FUNCTION_BLOCK FB3_XmlSvrRW_Recipe
VAR_INPUT
	bWriteSt				: BOOL;
	bReadSt					: BOOL;
	bShutdownRequestFlag 	: BOOL;

	eVariableType			: E_XMLVariableType;
	eXmlRwMode				: E_XmlRWMode;
		
	sDefaultFilePath		: STRING := 'C:\JKS\PLC\XML\';
	sFileExtension			: STRING := 'XML';
	
END_VAR
VAR_OUTPUT
	bWrite_Done				: BOOL;
	bWrite_Busy				: BOOL;
	bWrite_Error			: BOOL;
	udWrite_ErrId			: UDINT;
	bRead_Done				: BOOL;
	bRead_Busy				: BOOL;
	bRead_Error				: BOOL;
	udRead_ErrId 			: UDINT;
	bReadyToShutdownFlag 	: BOOL;
	sErrorMessage			: STRING;
	iTotalTime_100ms		: INT;
	iExportedImportedQty	: INT;
	iProgressPercentage		: INT;
END_VAR

VAR
		fbXmlSrvWriteByAdd	: FB_XmlSrvWrite;
		fbXmlSrvReadByAdd	: FB_XmlSrvRead;
		fbFileDelete		: FB_FileDelete;
	bWriteStRE						: R_TRIG;
	bReadStRE						: R_TRIG;
	iArrayId_ProRepRecipeQty		: INT;
	iArrayId_iSSERRecipeQty			: INT;
	iArrayId_iSSURRecipeQty			: INT;
	iArrayId_iSSMRRecipeQty			: INT;
	iArrayId_SSERProcessStnQty		: INT;
	iArrayId_SSURProcessStnQty		: INT;
	iArrayId_SSMRProcessStnQty		: INT;
	iFL								: INT;
	iCase							: INT;
	bFound							: BOOL;

	bWriteSt_Int					: BOOL;
	bReadSt_Int						: BOOL;
	bWrite_Busy_Int					: BOOL;
	bRead_Busy_Int					: BOOL;
	bFileDeleteSt					: BOOL;
	sFilePath_Int					: T_MaxString;
	sXPath_Int						: T_MaxString;

	
	iRepType			: INT;
	
	
	pSymAddr_Int		: PVOID;
	pSymAddr_Empty		: PVOID;

	cbSymSize_Int		: UDINT;
	sFileName_Main			: STRING;
	sFileName_Sub1			: STRING;
	sFileName_Sub2			: STRING;

	sXPath_Main			: STRING; 	// No Spacing is allowed
	sXPath_Sub1			: STRING;	// No Spacing is allowed
	sXPath_Sub2			: STRING;	// No Spacing is allowed

	
	bRead_Error_Int: BOOL;
	iTotalWriteTask: INT;
	iProRepTask: INT;
	iSSERTask: INT;
	iSSURTask: INT;
	iSSMRTask: INT;
END_VAR


IF NOT bWriteSt AND NOT bReadSt THEN
	iCase 	:= 0;
END_IF

bWriteStRE(CLK	:=bWriteSt AND NOT bShutdownRequestFlag 	, Q=> );
bReadStRE(CLK	:=bReadSt AND NOT bShutdownRequestFlag  	, Q=> );


// Shutdown request control
	bReadyToShutdownFlag := NOT bWrite_Busy AND NOT bRead_Busy AND bShutdownRequestFlag;


// Capture Total Time for Read or Write
IF iCase = 1 OR (iCase >= 10 AND iCase < 19) OR (iCase >= 20 AND iCase < 29) THEN
	IF bClockPulse_0_1Sec THEN
		iTotalTime_100ms := iTotalTime_100ms + 1;
	END_IF
END_IF


fbXmlSrvWriteByAdd(
	sNetId			:= '', 
	ePath			:= PATH_GENERIC, 
	nMode			:= XMLSRV_ADDMISSING, 
	pSymAddr		:= pSymAddr_Int, 
	cbSymSize		:= cbSymSize_Int, 
	sFilePath		:= sFilePath_Int, 
	sXPath			:= sXPath_Int, 
	bExecute		:= bWriteSt_Int, 
	tTimeout		:= T#5S, 
	bBusy			=> bWrite_Busy_Int, 
	bError			=> bWrite_Error);

fbXmlSrvReadByAdd(
	sNetId			:= '', 
	ePath			:= PATH_GENERIC, 
	nMode			:= XMLSRV_SKIPMISSING, 
	pSymAddr		:= pSymAddr_Int, 
	cbSymSize		:= cbSymSize_Int, 
	sFilePath		:= sFilePath_Int, 
	sXPath			:= sXPath_Int, 
	bExecute		:= bReadSt_Int, 
	tTimeout		:= T#5S, 
	bBusy			=> bRead_Busy_Int, 
	bError			=> bRead_Error_Int, 
	nErrId			=> );

IF 		bWriteStRE.Q 	AND NOT bReadSt 	AND NOT bRead_Busy 	THEN 	iCase := 1; 	bWrite_Busy := TRUE;
ELSIF	bReadStRE.Q		AND NOT bWriteSt 	AND NOT bWrite_Busy	THEN 	iCase := 1;		bRead_Busy := TRUE;			END_IF	

IF bRead_Error_Int AND fbXmlSrvReadByAdd.nErrId <> 1804 THEN
	bRead_Error := TRUE;
ELSE	
	bRead_Error := FALSE;
END_IF

CASE iCase OF
	
	0: 	// Reset ALL

			iArrayId_ProRepRecipeQty		:= 0;
			iArrayId_iSSERRecipeQty			:= 0;
			iArrayId_iSSURRecipeQty			:= 0;
			iArrayId_iSSMRRecipeQty			:= 0;
			iArrayId_SSERProcessStnQty		:= 0;
			iArrayId_SSURProcessStnQty		:= 0;
			iArrayId_SSMRProcessStnQty		:= 0;

			udWrite_ErrId			:= 0;
			bWrite_Busy				:= FALSE;
			bWrite_Error			:= FALSE;
			bWrite_Done				:= FALSE;

			udRead_ErrId			:= 0;
			bRead_Busy				:= FALSE;
			bRead_Error				:= FALSE;
			bRead_Done				:= FALSE;
	
			
			iTotalTime_100ms		:= 0;	

			bWriteSt_Int 			:= FALSE;
			bReadSt_Int 			:= FALSE;
			bFileDeleteSt			:= FALSE;
		
			iExportedImportedQty	:= 0;			
			pSymAddr_Int			:= pSymAddr_Empty;
			cbSymSize_Int			:= 0;	
			sFilePath_Int			:= '';
			sXPath_Int				:= '';	
			
			iRepType				:= 0;   // 1: Product Recipe, 2: SSER, 3: SSUR, 4: SSMR

			
			
			
	1: // Check Avaiable Array to trigger Read/Write

			IF iRepType 					< 1 	THEN iRepType 						:= 1; 	END_IF
			IF iArrayId_ProRepRecipeQty		< 1 	THEN iArrayId_ProRepRecipeQty	 	:= 1;	END_IF
			IF iArrayId_SSERProcessStnQty 	< 1 	THEN iArrayId_SSERProcessStnQty 	:= 1;	END_IF
			IF iArrayId_iSSERRecipeQty 		< 1	 	THEN iArrayId_iSSERRecipeQty 		:= 1; 	END_IF			
			IF iArrayId_SSURProcessStnQty 	< 1 	THEN iArrayId_SSURProcessStnQty 	:= 1;	END_IF
			IF iArrayId_iSSURRecipeQty 		< 1	 	THEN iArrayId_iSSURRecipeQty 		:= 1; 	END_IF
			IF iArrayId_SSMRProcessStnQty 	< 1 	THEN iArrayId_SSMRProcessStnQty 	:= 1;	END_IF
			IF iArrayId_iSSMRRecipeQty 		< 1	 	THEN iArrayId_iSSMRRecipeQty 		:= 1; 	END_IF
				
			CASE eXmlRwMode OF 
			
(*				eXmlMode_MergeAllByType:
						acMergeAllByType();							// ACTION			
*)						
				eXmlMode_SeperateByProductAndStation:			
						acSeperateByProductAndStation();			// ACTION
			
(*				eXmlMode_SeperateAll:			
						acSeperateAll();							// ACTION
*)
			END_CASE

						acGenerate_Filename_XPath();				// ACTION		
		
			IF 		bWrite_Busy AND iCase <> 19 THEN		
					iCase 	:= 12;					
			
			ELSIF 	bRead_Busy AND iCase <> 29 THEN		
					iCase 	:= 22;					
			END_IF			

				
	12: // Write Start

			bWriteSt_Int := TRUE;
	
			IF fbXmlSrvWriteByAdd.bExecute AND NOT fbXmlSrvWriteByAdd.bBusy AND NOT fbXmlSrvWriteByAdd.bError 
			AND 	fbXmlSrvWriteByAdd.pSymAddr		= pSymAddr_Int
			AND 	fbXmlSrvWriteByAdd.cbSymSize	= cbSymSize_Int	
			AND 	fbXmlSrvWriteByAdd.sFilePath 	= sFilePath_Int
			AND 	fbXmlSrvWriteByAdd.sXPath		= sXPath_Int		
			THEN	iCase := 13; // Write Done -> Proceed to clear FB to prepare for Next Cycle (Array) 
					iExportedImportedQty := iExportedImportedQty + 1;			
				
			ELSIF fbXmlSrvWriteByAdd.bExecute AND fbXmlSrvWriteByAdd.bError THEN
				udWrite_ErrId := fbXmlSrvWriteByAdd.nErrId;
				mtLogErrorId();
				iCase := 99;	// WRITE ERROR

				
			END_IF

	13: 	//  Write - prepare for Next Cycle (Array) 
			
			bWriteSt_Int := FALSE;
	
			IF NOT fbXmlSrvWriteByAdd.bExecute AND NOT fbXmlSrvWriteByAdd.bBusy  THEN
				iCase := 1; // Proceed to Next Cycle (Array) 
			END_IF
		
		
	19: // Write - All Done 
		
			bWrite_Busy 	:= FALSE;
			bWrite_Done 	:= TRUE;
			
	22: // Read Start

			bReadSt_Int := TRUE;
	
			IF 		fbXmlSrvReadByAdd.bExecute AND NOT fbXmlSrvReadByAdd.bBusy AND NOT fbXmlSrvReadByAdd.bError 
			AND 	fbXmlSrvReadByAdd.pSymAddr		= pSymAddr_Int
			AND 	fbXmlSrvReadByAdd.cbSymSize		= cbSymSize_Int
			AND 	fbXmlSrvReadByAdd.sFilePath 	= sFilePath_Int
			AND 	fbXmlSrvReadByAdd.sXPath		= sXPath_Int		
			THEN	iCase := 23; bFileDeleteSt := TRUE;	// Read Done -> Proceed to delete file and clear FB to prepare for Next Cycle (Array)			
					iExportedImportedQty := iExportedImportedQty + 1;			

			ELSIF fbXmlSrvReadByAdd.bExecute AND fbXmlSrvReadByAdd.bError AND fbXmlSrvReadByAdd.nErrId = 1804 
			THEN	iCase := 23; // Object Not Found -> Skipped and Proceed to clear FB to prepare for Next Cycle (Array)		
					
			ELSIF fbXmlSrvReadByAdd.bExecute AND fbXmlSrvReadByAdd.bError THEN
				udRead_ErrId := fbXmlSrvReadByAdd.nErrId;
				mtLogErrorId();
				iCase := 99;	// READ ERROR
			END_IF

	23:		// Delete file after read
			fbFileDelete(
			sNetId			:= '', 
			sPathName		:= sFilePath_Int, 
			ePath			:= PATH_GENERIC, 
			bExecute		:= bFileDeleteSt, 
			tTimeout		:= T#2S, 
			bBusy			=> , 
			bError			=> , 
			nErrId			=> );		

			IF fbFileDelete.bExecute AND NOT fbFileDelete.bBusy THEN
				bFileDeleteSt := FALSE;
			END_IF

			IF NOT fbFileDelete.bExecute AND NOT bFileDeleteSt THEN
				iCase := 24;	// Delete file done, proceed to clear FB to prepare for Next Cycle (Array)
			END_IF
			
	24: 	//  Read - prepare for Next Cycle (Array) 
			
			bReadSt_Int := FALSE;
	
			IF NOT fbXmlSrvReadByAdd.bExecute AND NOT fbXmlSrvReadByAdd.bBusy  THEN
				iCase := 1; // Proceed to Next Cycle (Array)
			END_IF
		
		
	29: // Read - All Done 
		
			bRead_Busy 	:= FALSE;
			bRead_Done 	:= TRUE;
		
	
	99: // Error
	
			bWriteSt_Int 	:= FALSE;
			bReadSt_Int 	:= FALSE;

END_CASE

// Progress Percentage
		IF NOT bWriteSt AND NOT bReadSt  THEN
			iProgressPercentage := 0;			

		ELSIF (bWriteSt AND NOT bWrite_Done) OR (bReadSt AND NOT bRead_Done) THEN
			acProgressPercentage();
		
		ELSIF (bWriteSt AND bWrite_Done) OR (bReadSt AND bRead_Done) THEN
			iProgressPercentage := 100;			
		END_IF

ACTION acGenerate_Filename_XPath:

		IF 		bWrite_Busy THEN		
		sFilePath_Int	:=	concat(sDefaultFilePath,	'Manual_Export'	);
		sFilePath_Int	:=	concat(sFilePath_Int,		'\'				);
		sFilePath_Int	:=	concat(sFilePath_Int,		sFileName_Main	);
		
		ELSIF 	bRead_Busy THEN		
		sFilePath_Int	:=	concat(sDefaultFilePath,	'Manual_Import'	);
		sFilePath_Int	:=	concat(sFilePath_Int,		'\'				);
		sFilePath_Int	:=	concat(sFilePath_Int,		sFileName_Main	);
		END_IF			
	
		IF sFileName_Sub1 <> '' THEN
		sFilePath_Int	:=	concat(sFilePath_Int,		'_'				);
		sFilePath_Int	:=	concat(sFilePath_Int,		sFileName_Sub1	);
		END_IF
		
		IF sFileName_Sub2 <> '' THEN
		sFilePath_Int	:=	concat(sFilePath_Int,		'_'				);
		sFilePath_Int	:=	concat(sFilePath_Int,		sFileName_Sub2	);
		END_IF
		
		sFilePath_Int	:=	concat(sFilePath_Int,		'.'				);
		sFilePath_Int	:=	concat(sFilePath_Int,		sFileExtension	);


							
		sXPath_Int		:=	concat('/Recipe/',		sXPath_Main		);

		IF sXPath_Sub1 <> '' THEN
		sXPath_Int		:=	concat(sXPath_Int,		'/ID'			);
		sXPath_Int		:=	concat(sXPath_Int,		sXPath_Sub1		);
		END_IF
		
		IF sXPath_Sub2 <> '' THEN
		sXPath_Int		:=	concat(sXPath_Int,		'/ID'			);
		sXPath_Int		:=	concat(sXPath_Int,		sXPath_Sub2		);
		END_IF
END_ACTION

ACTION acMergeAllByType:

	IF 		iRepType 		= eXmlParTypeSSER                       
	THEN	pSymAddr_Int 	:= ADR	(fbMainStationProcess_Stn);  
			cbSymSize_Int	:= SIZEOF(fbMainStationProcess_Stn);
			sFileName_Main	:= 'MergeAll\SSER';                 
			sFileName_Sub1	:= 'All';                           
			sFileName_Sub2	:= '';                              
			sXPath_Main		:= 'AR2dsSSER';                       
			sXPath_Sub1		:= '';                                
			sXPath_Sub2		:= '';                                

			
	ELSIF 	iRepType 		= eXmlParTypeSSUR                       
	THEN	pSymAddr_Int 	:= ADR	(fbMainStationProcess_Stn);  
			cbSymSize_Int	:= SIZEOF(fbMainStationProcess_Stn);
			sFileName_Main	:= 'MergeAll\SSUR';                 
			sFileName_Sub1	:= 'All';                           
			sFileName_Sub2	:= '';                              
			sXPath_Main		:= 'AR2dsSSUR';                       
			sXPath_Sub1		:= '';                                
			sXPath_Sub2		:= '';     
			


	

	ELSE  	// All Done
			IF 		bWrite_Busy	THEN
				iCase 	:= 19;
			ELSIF 	bRead_Busy	THEN
				iCase 	:= 29;
			END_IF
	END_IF

	iRepType := iRepType +1;
END_ACTION

ACTION acProgressPercentage:

IF 		eXmlRwMode = eXmlMode_MergeAllByType THEN

		iTotalWriteTask 	:= 4; // Refer to E_XmlParType
		
		IF iRepType-1 >= 1 AND iRepType-1 <= 4 THEN 
			iProgressPercentage := ((iRepType-1)*100) / iTotalWriteTask;
		END_IF

		IF iProgressPercentage > 100 THEN iProgressPercentage := 100; END_IF
		
ELSIF	eXmlRwMode = eXmlMode_SeperateByProductAndStation THEN

		iProRepTask			:= C_iProRepRecipeQty;
		iSSERTask			:= C_iProcessStnQty;
		iSSURTask			:= C_iProcessStnQty;
		iSSMRTask			:= C_iProcessStnQty;
				
		iTotalWriteTask 	:= (iProRepTask) + (iSSERTask) + (iSSURTask) + (iSSMRTask);

			IF 		iRepType = eXmlParTypeProductRecipe THEN
						iProgressPercentage := (iArrayId_ProRepRecipeQty*100) / iTotalWriteTask;
			ELSIF 	iRepType = eXmlParTypeSSER THEN		
						iProgressPercentage := (iArrayId_iSSERRecipeQty*100) / iTotalWriteTask;
						iProgressPercentage := iProgressPercentage + ((iProRepTask*100) / iTotalWriteTask);
			ELSIF 	iRepType = eXmlParTypeSSUR THEN		
						iProgressPercentage := (iArrayId_iSSURRecipeQty*100) / iTotalWriteTask;
						iProgressPercentage := iProgressPercentage + ((iProRepTask*100) / iTotalWriteTask);
						iProgressPercentage := iProgressPercentage + ((iSSERTask*100) / iTotalWriteTask);
		(*	ELSIF 	iRepType = eXmlParTypeSSMR THEN		
						iProgressPercentage := (iArrayId_iSSMRRecipeQty*100) / iTotalWriteTask;
						iProgressPercentage := iProgressPercentage + ((iProRepTask*100) / iTotalWriteTask);
						iProgressPercentage := iProgressPercentage + ((iSSERTask*100) / iTotalWriteTask);
						iProgressPercentage := iProgressPercentage + ((iSSURTask*100) / iTotalWriteTask);
		*)				
			END_IF

			IF iProgressPercentage > 100 THEN iProgressPercentage := 100; END_IF
			
	
ELSIF	eXmlRwMode = eXmlMode_SeperateAll THEN

		iProRepTask			:= C_iProRepRecipeQty;
		iSSERTask			:= C_iProcessStnQty*C_iSSERRecipeQty;
		iSSURTask			:= C_iProcessStnQty*C_iSSURRecipeQty;
		iSSMRTask			:= C_iProcessStnQty*C_iSSMRRecipeQty;
				
		iTotalWriteTask 	:= (iProRepTask) + (iSSERTask) + (iSSURTask) + (iSSMRTask);

			IF 		iRepType = eXmlParTypeProductRecipe THEN
						iProgressPercentage := (iArrayId_ProRepRecipeQty*100) / iTotalWriteTask;
			ELSIF 	iRepType = eXmlParTypeSSER THEN		

						iProgressPercentage := ((((iArrayId_SSERProcessStnQty-1)*C_iSSERRecipeQty) + iArrayId_iSSERRecipeQty) *100) / iTotalWriteTask;
						iProgressPercentage := iProgressPercentage + ((iProRepTask*100) / iTotalWriteTask);

			ELSIF 	iRepType = eXmlParTypeSSUR THEN		
						iProgressPercentage := ((((iArrayId_SSURProcessStnQty-1)*C_iSSURRecipeQty) + iArrayId_iSSURRecipeQty) *100) / iTotalWriteTask;
						iProgressPercentage := iProgressPercentage + ((iProRepTask*100) / iTotalWriteTask);
						iProgressPercentage := iProgressPercentage + ((iSSERTask*100) / iTotalWriteTask);
		(*	ELSIF 	iRepType = eXmlParTypeSSMR THEN		
						iProgressPercentage := ((((iArrayId_SSMRProcessStnQty-1)*C_iSSMRRecipeQty) + iArrayId_iSSMRRecipeQty) *100) / iTotalWriteTask;
						iProgressPercentage := iProgressPercentage + ((iProRepTask*100) / iTotalWriteTask);
						iProgressPercentage := iProgressPercentage + ((iSSERTask*100) / iTotalWriteTask);
						iProgressPercentage := iProgressPercentage + ((iSSURTask*100) / iTotalWriteTask);
		*)				
			END_IF

			IF iProgressPercentage > 100 THEN iProgressPercentage := 100; END_IF
		
END_IF
END_ACTION

ACTION acSeperateByProductAndStation:

	IF 		iRepType = eXmlParTypeSSER 	THEN				
			
            	pSymAddr_Int 	:= ADR		(fbMainStationProcess_Stn[iArrayId_SSERProcessStnQty].StnSeqProcessfb.fbStationSequenceRecipefb.ARDsStorageStationSequenceRecipeMemory);
				cbSymSize_Int	:= SIZEOF	(fbMainStationProcess_Stn[iArrayId_SSERProcessStnQty].StnSeqProcessfb.fbStationSequenceRecipefb.ARDsStorageStationSequenceRecipeMemory);
				sFileName_Main	:= 'ByProductAndStation\SSER';
				sFileName_Sub1	:= TO_STRING(iArrayId_SSERProcessStnQty);
				sFileName_Sub2	:= ''; 
				sXPath_Main		:= 'AR2dsSSER';
				sXPath_Sub1		:= TO_STRING(iArrayId_SSERProcessStnQty);
				sXPath_Sub2		:= '';
			
			IF 		iArrayId_SSERProcessStnQty + 1 > C_iProcessStnQty THEN 
					iRepType 					:= iRepType +1;
            		iArrayId_SSERProcessStnQty 	:= 1;
			ELSE
					iArrayId_SSERProcessStnQty 	:= iArrayId_SSERProcessStnQty + 1;
			END_IF
			

			
			
	ELSIF	iRepType = eXmlParTypeSSUR	THEN

					pSymAddr_Int 	:= ADR		(fbMainStationProcess_Stn[iArrayId_SSURProcessStnQty].StnSeqProcessfb.fbStationSubRecipefb);
					cbSymSize_Int	:= SIZEOF	(fbMainStationProcess_Stn[iArrayId_SSURProcessStnQty].StnSeqProcessfb.fbStationSubRecipefb);
					sFileName_Main	:= 'ByProductAndStation\SSUR';
					sFileName_Sub1	:= TO_STRING(iArrayId_SSURProcessStnQty);
					sFileName_Sub2	:= '';
					sXPath_Main		:= 'AR2dsSSUR';
					sXPath_Sub1		:= TO_STRING(iArrayId_SSURProcessStnQty);
					sXPath_Sub2		:= '';

			IF 		iArrayId_SSURProcessStnQty + 1 > C_iProcessStnQty THEN 
					iRepType 					:= iRepType +1;
					iArrayId_SSURProcessStnQty 	:= 1;
			ELSE
					iArrayId_SSURProcessStnQty 	:= iArrayId_SSURProcessStnQty + 1;
			END_IF

			
	ELSIF 	iRepType = eXmlParTypeProductRecipe	THEN
					
					pSymAddr_Int 	:= ADR		(PnPstorageMemory_Arm.fbGnrProductRecipeMemory_Main.fbA1PnpSequenceMemory.ARDsPnpSequenceMemory[iArrayId_ProRepRecipeQty]);
					cbSymSize_Int	:= SIZEOF	(PnPstorageMemory_Arm.fbGnrProductRecipeMemory_Main.fbA1PnpSequenceMemory.ARDsPnpSequenceMemory[iArrayId_ProRepRecipeQty]);
					sFileName_Main	:= 'ByProductAndStation\ProductRecipe';
					sFileName_Sub1	:= TO_STRING(iArrayId_ProRepRecipeQty);
					sFileName_Sub2	:= '';
					sXPath_Main		:= 'ARdsProductRecipe';
					sXPath_Sub1		:= TO_STRING(iArrayId_ProRepRecipeQty);
					sXPath_Sub2		:= '';

			IF 		iArrayId_ProRepRecipeQty + 1 > C_iProRepRecipeQty THEN 
					iRepType 					:= iRepType +1;
					iArrayId_ProRepRecipeQty 	:= 1;
			ELSE				
					iArrayId_ProRepRecipeQty 	:= iArrayId_ProRepRecipeQty + 1; 
			END_IF			
			

		ELSE	// All Done
				IF 		bWrite_Busy	THEN
					iCase 	:= 19;
				ELSIF 	bRead_Busy	THEN
					iCase 	:= 29;
				END_IF
		
		END_IF
END_ACTION

METHOD PRIVATE mtLogErrorId : BOOL
VAR_INPUT
	
END_VAR
		IF 		bWriteSt_Int 
		THEN	sErrorMessage := concat('XML Write Error -' , 	'ErrorId: ');
				sErrorMessage := concat (sErrorMessage, 		TO_STRING(udWrite_ErrId));
				sErrorMessage := concat (sErrorMessage, 		' - ');
				sErrorMessage := concat (sErrorMessage, 		sFilePath_Int);
		ELSIF	bReadSt_Int
		THEN	sErrorMessage := concat('XML Read Error -' , 	'ErrorId: ');
				sErrorMessage := concat (sErrorMessage, 		TO_STRING(udRead_ErrId));
				sErrorMessage := concat (sErrorMessage, 		' - ');
				sErrorMessage := concat (sErrorMessage, 		sFilePath_Int);
		END_IF
	
		mtLogErrorId := TRUE;
END_METHOD

END_FUNCTION_BLOCK

(* stored: Version 1.1.0.1, ProductVersion 3.1.4024.12
   POU FB3_XmlSvrRW_Recipe: Id {0e2888df-b51a-44bd-aa41-62eb0ce64752}, SpecialFunc None
   Action acGenerate_Filename_XPath: Id {578d48be-11b2-4d76-a275-8b5af124aa9b}
   Action acMergeAllByType: Id {b07ef4d2-a83c-49a9-9329-2fb15ff5fd15}
   Action acProgressPercentage: Id {b8ce1557-5292-4f15-9b5e-e664bee9f8d1}
   Action acSeperateByProductAndStation: Id {530cc17b-b3e2-4c27-8478-922e1b17f33e}
   Method mtLogErrorId: Id {e3dd4cd3-e98c-472b-a116-4816a765003f} *)
